(* Logix 5000 project; controller APM_ejercicio_1 vendor 1 type 14 code 156 rev 32.11; software revision 32.00 *)

TASK MainTask (continuous, watchdog 500 ms) : MainProgram, Flancos_Sensores

MODULES
   Local : vendor 1 type 14 code 156 (Compact 0, rev 32.11)
      Entradas_Digitales : 1769-IQ16 (Compact 4, rev 1.1, Input RPI 20 ms)
      Salidas_Digitales : vendor 1 type 7 code 86 (Compact 5, rev 2.1, Output RPI 20 ms)
      Variador_139 : PowerFlex 525-EENET (Ethernet 10.203.3.139, rev 5.1, Output RPI 20 ms)
END_MODULES

VAR_GLOBAL   (* controller tags *)
   AUX_1 : BOOL;
   AUX_2 : BOOL;
   AUX_3 : BOOL;
   AUX_4 : BOOL;
   AUX_5 : BOOL;
   AUX_6 : BOOL;
   AUX_7 : BOOL;
   Banda_2 : BOOL := 1;
   Bandera_1 : BOOL;
   Bandera_Funcionamiento : BOOL;
   Bit_aux : BOOL;
   BTN_E1 : BOOL;
   BTN_E2 : BOOL;
   BTN_E3 : BOOL;
   BTN_E4 : BOOL;
   BTN_E5 : BOOL;
   BTN_E6 : BOOL;
   BTN_PE1 : BOOL;
   BTN_PE2 : BOOL;
   BTN_PE3 : BOOL;
   BTN_PE4 : BOOL;
   BTN_PE5 : BOOL;
   BTN_PE6 : BOOL;
   Contador_E1 : COUNTER;
   Contador_E2 : COUNTER;
   Contador_E3 : COUNTER;
   Contador_E4 : COUNTER;
   Contador_E5 : COUNTER;
   Contador_E6 : COUNTER;
   Counter_Aux : COUNTER := (PRE := 2);
   CYCL_INI : BOOL;
   E1 : BOOL;
   E2 : BOOL;
   E3 : BOOL;
   E4 : BOOL;
   Estacion_1 : BOOL;
   Estacion_2 : BOOL;
   Estacion_3 : BOOL;
   Estacion_4 : BOOL;
   Estacion_5 : BOOL;
   Estacion_6 : BOOL;
   Estacion_INI : BOOL;
   FS_CHNG_OK : BOOL;
   FS_E1 : BOOL;
   FS_E2 : BOOL;
   FS_E3 : BOOL;
   FS_E4 : BOOL;
   FS_E5 : BOOL;
   FS_E6 : BOOL;
   MTR_STOP : BOOL;
   NUM_BCYCL : INT;
   NUM_BCYCL_0 : DINT;
   NUM_BCYCL_1 : DINT;
   NUM_BCYCL_2 : DINT;
   NUM_BCYCL_TOTAL : DINT;
   Pantallas : BOOL;
   Process_ON : BOOL := 1;
   Producto : INT;
   Producto_1 : DINT;
   Producto_3 : DINT;
   Producto_6 : DINT;
   S_CHNG_OK : BOOL;
   S_E1 : BOOL;
   S_E2 : BOOL;
   S_E3 : BOOL;
   S_E4 : BOOL;
   S_E5 : BOOL;
   S_E6 : BOOL;
   START : ALIAS FOR Local:4:I.Data.0;
   T1 : BOOL;
   T2 : BOOL;
   T3 : BOOL;
   T4 : BOOL;
   TT1 : BOOL;
   Var_aux : REAL := 3600.0;
   Velocidad_Banda : DINT := 6;
END_VAR

PROGRAM Flancos_Sensores   (* main routine MainRoutine *)

ROUTINE Flancos_y_Contadores   (* ladder *)
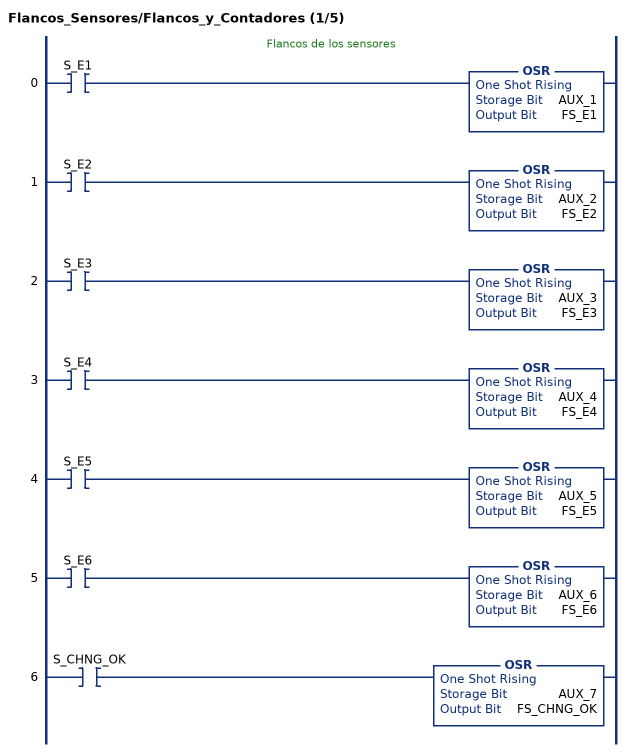
   // Flancos de los sensores
   0: XIC(S_E1)OSR(AUX_1,FS_E1);
   1: XIC(S_E2)OSR(AUX_2,FS_E2);
   2: XIC(S_E3)OSR(AUX_3,FS_E3);
   3: XIC(S_E4)OSR(AUX_4,FS_E4);
   4: XIC(S_E5)OSR(AUX_5,FS_E5);
   5: XIC(S_E6)OSR(AUX_6,FS_E6);
   6: XIC(S_CHNG_OK)OSR(AUX_7,FS_CHNG_OK);
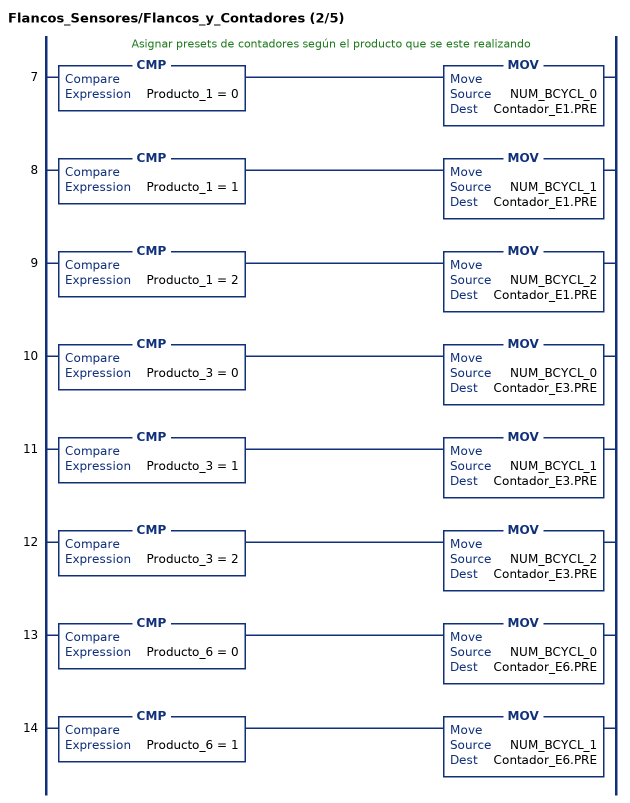
   // Asignar presets de contadores según el producto que se este realizando
   7: CMP(Producto_1 = 0)MOV(NUM_BCYCL_0,Contador_E1.PRE);
   8: CMP(Producto_1 = 1)MOV(NUM_BCYCL_1,Contador_E1.PRE);
   9: CMP(Producto_1 = 2)MOV(NUM_BCYCL_2,Contador_E1.PRE);
   10: CMP(Producto_3 = 0)MOV(NUM_BCYCL_0,Contador_E3.PRE);
   11: CMP(Producto_3 = 1)MOV(NUM_BCYCL_1,Contador_E3.PRE);
   12: CMP(Producto_3 = 2)MOV(NUM_BCYCL_2,Contador_E3.PRE);
   13: CMP(Producto_6 = 0)MOV(NUM_BCYCL_0,Contador_E6.PRE);
   14: CMP(Producto_6 = 1)MOV(NUM_BCYCL_1,Contador_E6.PRE);
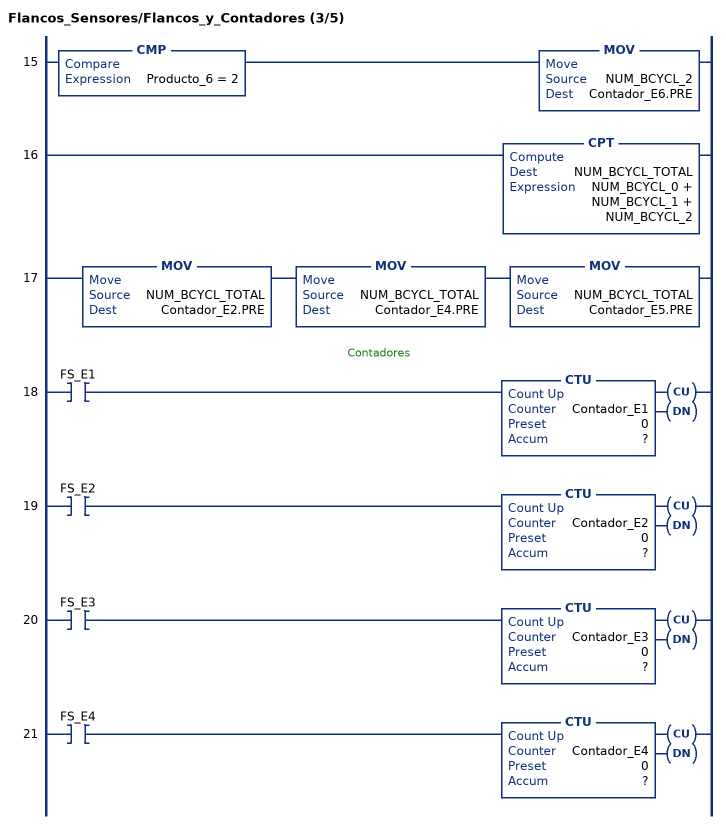
   15: CMP(Producto_6 = 2)MOV(NUM_BCYCL_2,Contador_E6.PRE);
   16: CPT(NUM_BCYCL_TOTAL,NUM_BCYCL_0 + NUM_BCYCL_1 + NUM_BCYCL_2);
   17: MOV(NUM_BCYCL_TOTAL,Contador_E2.PRE)MOV(NUM_BCYCL_TOTAL,Contador_E4.PRE)MOV(NUM_BCYCL_TOTAL,Contador_E5.PRE);
   // Contadores
   18: XIC(FS_E1)CTU(Contador_E1,?,?);
   19: XIC(FS_E2)CTU(Contador_E2,?,?);
   20: XIC(FS_E3)CTU(Contador_E3,?,?);
   21: XIC(FS_E4)CTU(Contador_E4,?,?);
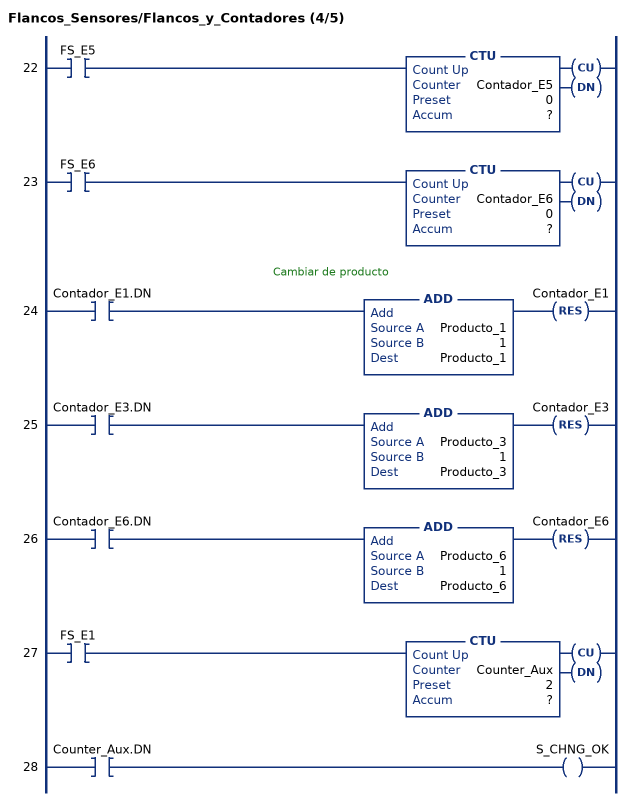
   22: XIC(FS_E5)CTU(Contador_E5,?,?);
   23: XIC(FS_E6)CTU(Contador_E6,?,?);
   // Cambiar de producto
   24: XIC(Contador_E1.DN)ADD(Producto_1,1,Producto_1)RES(Contador_E1);
   25: XIC(Contador_E3.DN)ADD(Producto_3,1,Producto_3)RES(Contador_E3);
   26: XIC(Contador_E6.DN)ADD(Producto_6,1,Producto_6)RES(Contador_E6);
   27: XIC(FS_E1)CTU(Counter_Aux,?,?);
   28: XIC(Counter_Aux.DN)OTE(S_CHNG_OK);
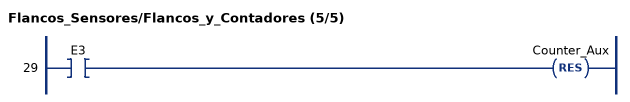
   29: XIC(E3)RES(Counter_Aux);
END_ROUTINE

ROUTINE MainRoutine   (* ladder *)
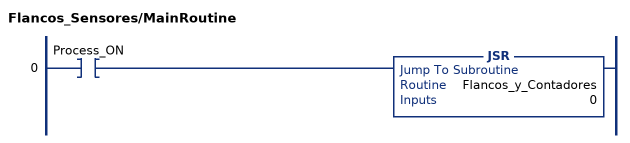
   0: XIC(Process_ON)JSR(Flancos_y_Contadores,0);
END_ROUTINE
END_PROGRAM

PROGRAM MainProgram   (* main routine MainRoutine *)

ROUTINE Logica_Parte_2   (* ladder *)
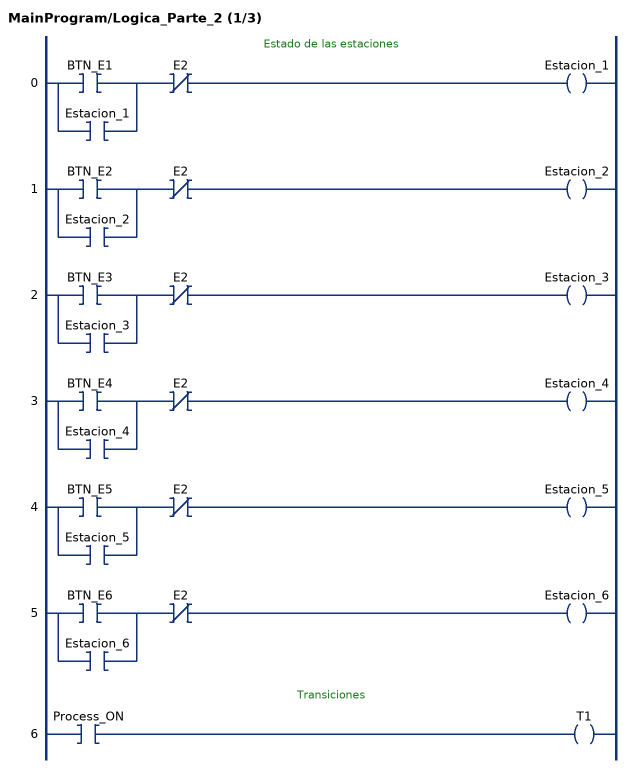
   // Estado de las estaciones
   0: [XIC(BTN_E1) ,XIC(Estacion_1) ]XIO(E2)OTE(Estacion_1);
   1: [XIC(BTN_E2) ,XIC(Estacion_2) ]XIO(E2)OTE(Estacion_2);
   2: [XIC(BTN_E3) ,XIC(Estacion_3) ]XIO(E2)OTE(Estacion_3);
   3: [XIC(BTN_E4) ,XIC(Estacion_4) ]XIO(E2)OTE(Estacion_4);
   4: [XIC(BTN_E5) ,XIC(Estacion_5) ]XIO(E2)OTE(Estacion_5);
   5: [XIC(BTN_E6) ,XIC(Estacion_6) ]XIO(E2)OTE(Estacion_6);
   // Transiciones
   6: XIC(Process_ON)OTE(T1);
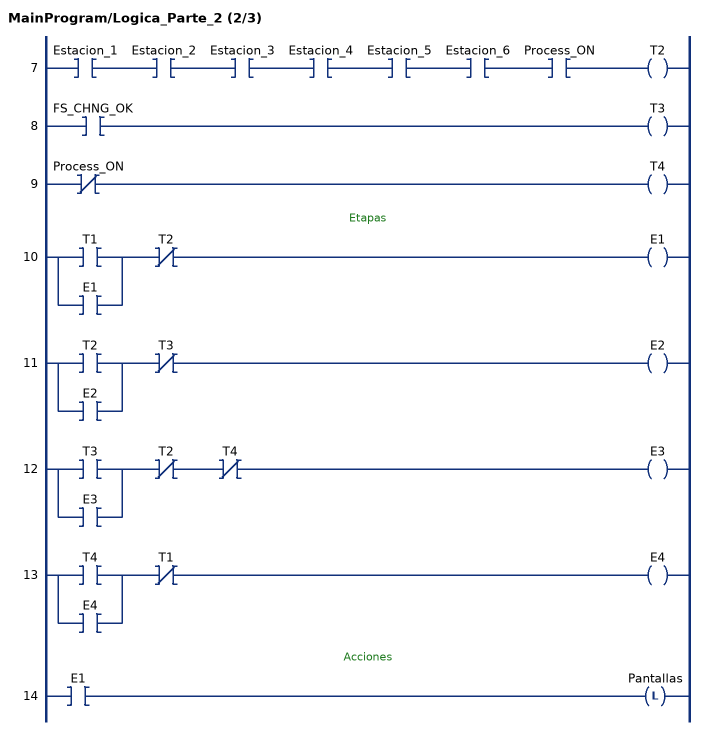
   7: XIC(Estacion_1)XIC(Estacion_2)XIC(Estacion_3)XIC(Estacion_4)XIC(Estacion_5)XIC(Estacion_6)XIC(Process_ON)OTE(T2);
   8: XIC(FS_CHNG_OK)OTE(T3);
   9: XIO(Process_ON)OTE(T4);
   // Etapas
   10: [XIC(T1) ,XIC(E1) ]XIO(T2)OTE(E1);
   11: [XIC(T2) ,XIC(E2) ]XIO(T3)OTE(E2);
   12: [XIC(T3) ,XIC(E3) ]XIO(T2)XIO(T4)OTE(E3);
   13: [XIC(T4) ,XIC(E4) ]XIO(T1)OTE(E4);
   // Acciones
   14: XIC(E1)OTL(Pantallas);
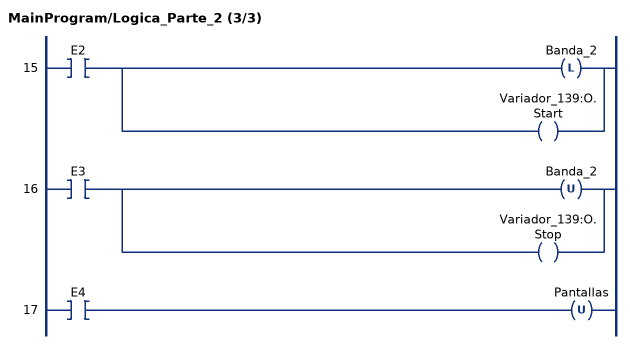
   15: XIC(E2)[OTL(Banda_2) ,OTE(Variador_139:O.Start) ];
   16: XIC(E3)[OTU(Banda_2) ,OTE(Variador_139:O.Stop) ];
   17: XIC(E4)OTU(Pantallas);
END_ROUTINE

ROUTINE MainRoutine   (* ladder *)
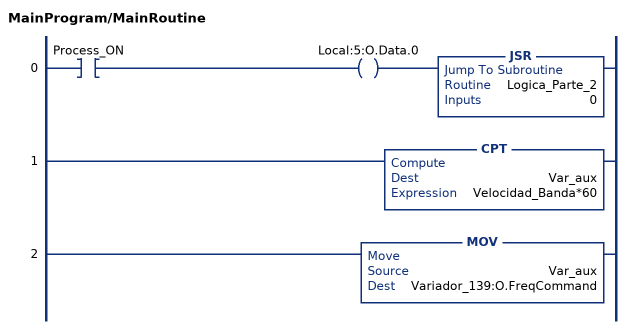
   0: XIC(Process_ON)OTE(Local:5:O.Data.0)JSR(Logica_Parte_2,0);
   1: CPT(Var_aux,Velocidad_Banda*60);
   2: MOV(Var_aux,Variador_139:O.FreqCommand);
END_ROUTINE
END_PROGRAM
